PROGRAM P_FunctionGenerators
VAR
	
nPositionAr: ARRAY [0..2, 0..999]  OF LREAL; ///1000 positions to fill 1 second, 3 seconds worth of buffer. position data in ms.
timer: TON; //track time
ElapsedTIME :TIME;
nPostionTarget: LREAL;
nCase: INT;

END_VAR

CASE nCase OF
	1://Random inputs within 10 of each other
	2://
	3://
	4://
	
END_CASE

END_PROGRAM

(* stored: Version 1.1.0.1, ProductVersion 3.1.4024.3
   POU P_FunctionGenerators: Id {115fcafb-7e59-4bfc-a156-7bd475b390a7}, SpecialFunc None *)
